PROGRAM z_TEMP

VAR
	rOutRegTemp: REAL;
END_VAR

(*-------------------------------------------------------------------------------------------------------*)
(*v061  Valvula de vapor*)
mc._02_TEMP.v061_Steam.xOpen:= F_TERMOREG.Z_xVapor OR
								F_ISOTERMA.Z_xVapor;

(*-------------------------------------------------------------------------------------------------------*)
(*v062  Valvula de enfriamiento*)
mc._02_TEMP.v062_Cool.xOpen:= F_TERMOREG.z_xEnfria OR
								F_ISOTERMA.z_xEnfria;

(*-------------------------------------------------------------------------------------------------------*)
(*v060  Apertura ValvulaModulante*)
//calentar temo
IF Mc._02_TEMP.v061_Steam.xOpen AND F_TERMOREG.xActv THEN
	Mc._02_TEMP.v060_Aper.rValue:= F_TERMOREG.z_rApertVapor;
END_IF

//calentar ISOTERMA
IF Mc._02_TEMP.v061_Steam.xOpen AND F_ISOTERMA.xActv THEN
	mc._02_TEMP.v060_Aper.rValue:= F_ISOTERMA.z_rApertVapor;
END_IF

//ENFRIAR TERMO
IF Mc._02_TEMP.v062_Cool.xOpen AND F_TERMOREG.xActv THEN
	MC._02_TEMP.v060_Aper.rValue:= F_TERMOREG.z_rApertEnfria;
END_IF

//ENFRIAR ISOTERMA
IF
	MC._02_TEMP.v062_Cool.xOpen AND F_ISOTERMA.xActv THEN
	MC._02_TEMP.v060_Aper.rValue:= F_ISOTERMA.z_rApertEnfria;
END_IF

//OUTPUT Regulacion Temperatura

rOutRegTemp:= Canvi_Escala(
				In:= mc._02_TEMP.v060_Aper.rValue, 
				In_Min:= 0, 
				In_Max:= 1, 
				Out_Min:= 0, 
				Out_Max:= 32675);
	

(*-------------------------------------------------------------------------------------------------------*)
(*v063 Retorno condensados*)
mc._02_TEMP.v063_RetCon.xOpen:= F_TERMOREG.z_xRetonoCond;

(*-------------------------------------------------------------------------------------------------------*)

END_PROGRAM

(* stored: Version 1.1.0.1, ProductVersion 3.1.4024.10
   POU z_TEMP: Id {2c3a6b58-e97e-46d4-9892-884ea7f1ceec}, SpecialFunc None *)
